FUNCTION TFCheckPalletFull : INT
VAR_INPUT
	WorkArea : POINTER TO ARRAY [1..MAXAREA] OF TFMachinePalletizer_WorkArea;
	WorkAreaState : POINTER TO ARRAY [1..MAXAREA] OF TFMachinePalletizer_WorkAreaState;
	//PX_WorkArea : ARRAY [1..MAXAREA] OF BOOL;
	WorkPickPointState : POINTER TO ARRAY [1..MAXPICKPOINT] OF TFMachinePalletizer_WorkPickPointState;
	Forming : POINTER TO ARRAY [1..MAXFORMING] OF TFMachinePalletizer_Forming;
END_VAR
VAR
	i : INT;
	k : INT;
END_VAR

TFCheckPalletFull := 0;
FOR k := 1 TO MAXPICKPOINT DO
	//IF WorkPickPointState^[k].State = 1 THEN
		FOR i:=1 TO MAXAREA DO	
			IF WorkArea^[i].Enable = 1 AND WorkArea^[i].Typology = TYPOLOGY_PALLET AND 
				WorkArea^[i].Code = 0  AND 
				//WorkAreaState^[i].State <= WORKAREA_STATE_OCCUPIED_WORKING AND 
				(Forming^[WorkAreaState^[i].F].PackXP[WorkAreaState^[i].P].Grip <> -1 OR 
				Forming^[WorkAreaState^[i].F].PackXN[WorkAreaState^[i].P].Grip <> -1) THEN
				RETURN;
			END_IF
		END_FOR
	//ELSE
	//	;//RETURN;	
	//END_IF	
END_FOR	
	
TFCheckPalletFull := 1;

END_FUNCTION

(* stored: Version 1.1.0.1, ProductVersion 3.1.4024.11
   POU TFCheckPalletFull: Id {332d31e2-cd79-4f58-b678-78ea0f4f90cd}, SpecialFunc None *)
